// TIA Portal V20 export
// export: Created 2025-12-01T14:57:05.3084144Z, ExportSetting None, DisplayName Totally Integrated Automation Portal, DisplayVersion V20 Update 3, DisplayName TIA Portal Openness, DisplayVersion V20 Update 3, DisplayName TIA Portal Version Control Interface, DisplayVersion V20 Update 3, DisplayName STEP 7 Professional, DisplayVersion V20 Update 3, DisplayName STEP 7 Safety, DisplayVersion V20 Update 2, DisplayName WinCC Basic/Comfort/Advanced, DisplayVersion V20 Update 3, DisplayName WinCC Professional, DisplayVersion V20 Update 3, DisplayName WinCC Unified, DisplayVersion V20 Update 3
FUNCTION "FC775_Altura_PilaDeCajasPlastico" : Void   // FC775, STL
TITLE = Activacion de la Guias del Apilador y Desapilador de Cajas
{ S7_Optimized_Access := 'FALSE' }
AUTHOR : TRACKING
NAME : 20130301
VERSION : 3.0
// stored: AutoNumber false
   VAR_INPUT
      Mesa : UInt;   // Numero de Mesa
      AlturaActivarGuias : UInt;   // Altura a Activar las Guias
   END_VAR
   VAR_OUTPUT
      ActivarGuias : Bool;   // Activar las Guias
   END_VAR
   VAR_TEMP
      NumeroUT : UInt;   // Numero de UT
      AlturaPilaActual : UInt;   // Altura de la Pila de las UTs en la Mesa
   END_VAR
BEGIN

NETWORK
TITLE = Inicialializar
////////////////////////////////////////////////////////////////////////////
// --- Inicializar variables

      SET;
      R     #ActivarGuias;  // Desactivar Salida
      L     0;  // Calculo de la Altura de la Pila
      T     #AlturaPilaActual;



NETWORK
TITLE = Calculo de Activacion
////////////////////////////////////////////////////////////////////////////
// --- Ver si hay UT's en la Mesa


      L     "DB810_ColasMesas".Colas[#Mesa].UT_PrimeraMesa;
      T     #NumeroUT;

      L     #NumeroUT;  // Si no hay UT's
      L     0;
      ==I;
      JC    Final;


////////////////////////////////////////////////////////////////////////////
// --- Recorrer la Cola de la Mesa
// --- Calcular la Altura que tiene la Pila de UT's

Inicio_BucleMesa:NOP   0;

      L     #AlturaPilaActual;  // Sumar la Altura de la UT a la Pila
      L     "DB815_UTs_Datos".UT[#NumeroUT].CotaAltura;
      +I;
      T     #AlturaPilaActual;

      L     "DB812_UTs_Control".UT[#NumeroUT].UT_SiguienteMesa;
      T     #NumeroUT;

      L     #NumeroUT;
      L     0;
      <>I;
      JC    Inicio_BucleMesa;  // Quedan UT's en la Mesa ?


////////////////////////////////////////////////////////////////////////////
// --- Comparar para ver si hay que activar las Guias

      L     #AlturaPilaActual;
      L     #AlturaActivarGuias;
      <I;
      JC    Final;

// --- El Mayor la Altura de las UT's de la Mesa
// --- Activar la salida

      S     #ActivarGuias;



NETWORK
TITLE = Final de la Funcion
////////////////////////////////////////////////////////////////////////////
// --- Final de la Función
Final:NOP   0;


END_FUNCTION
